Staubli VAL3: Bewegungsattribute.pjx

--- Bewegungsattribute.pjx ---
Parameters version=s7.5.3 stackSize=5000 millimeterUnit=true
Program file=MoveJoint.pgx
Program file=MoveLine.pgx
Program file=start.pgx
Program file=stop.pgx
Program file=main.pgx
Data file=Bewegungsattribute.dtx

--- Bewegungsattribute.dtx ---
frame StaubliTX240Base = {x=0.000, y=0.000, z=0.000, rx=-0.000, ry=0.000, rz=-0.000, fatherId=world[0]}
tool tCurrentTool = {x=0.000, y=0.000, z=0.000, rx=-0.000, ry=0.000, rz=-0.000, fatherId=flange[0]}
mdesc mCurrentSpeed
pointRx pPointRx1 = {}
pointRx pPointRx2 = {}

--- main.pgx ---
program main()
begin
    pPointRx1.config.shoulder = lefty
    pPointRx1.config.elbow = epositive
    pPointRx1.config.wrist = wpositive
    pPointRx2.config.shoulder = lefty
    pPointRx2.config.elbow = epositive
    pPointRx2.config.wrist = wpositive
    mCurrentSpeed.tvel = 100.00
    mCurrentSpeed.blend = joint
    mCurrentSpeed.reach = 0.010
    mCurrentSpeed.leave = 0.010
    		// Program Bewegungsattribute start
		// Program generated by RoboDK v5.2.1 for Staubli TX2-40 on 26/04/2021 13:26:34
		mCurrentSpeed.accel = 30.000
		mCurrentSpeed.decel = 30.000
		mCurrentSpeed.vel = 30.000
		mCurrentSpeed.tvel = 30.000
		mCurrentSpeed.rvel = 30.000
		link(pPointRx1,StaubliTX240Base)
		link(pPointRx2,StaubliTX240Base)
		call MoveJoint(0.00000,0.00000,90.00000,0.00000,0.00000,-0.00000)
		call MoveJoint(0.75339,44.25550,52.41940,0.00000,83.32510,0.75339)
		call MoveJoint(-10.97790,47.35230,41.99440,0.00000,90.65320,-10.97790)
		call MoveJoint(-1.36528,60.04990,34.36770,0.00000,85.58250,-1.36528)
		call MoveJoint(0.00000,0.00000,90.00000,0.00000,0.00000,-0.00000)
		mCurrentSpeed.rvel = 1000.000
		call MoveJoint(0.75339,44.25550,52.41940,0.00000,83.32510,0.75339)
		call MoveJoint(-10.97790,47.35230,41.99440,0.00000,90.65320,-10.97790)
		call MoveJoint(-1.36528,60.04990,34.36770,0.00000,85.58250,-1.36528)
		call MoveJoint(0.00000,0.00000,90.00000,0.00000,0.00000,-0.00000)
		mCurrentSpeed.tvel = 1000.000
		call MoveJoint(0.75339,44.25550,52.41940,0.00000,83.32510,0.75339)
		call MoveJoint(-10.97790,47.35230,41.99440,0.00000,90.65320,-10.97790)
		call MoveJoint(-1.36528,60.04990,34.36770,0.00000,85.58250,-1.36528)
		call MoveJoint(0.00000,0.00000,90.00000,0.00000,0.00000,-0.00000)
		mCurrentSpeed.vel = 100.000
		call MoveJoint(0.75339,44.25550,52.41940,0.00000,83.32510,0.75339)
		call MoveJoint(-10.97790,47.35230,41.99440,0.00000,90.65320,-10.97790)
		call MoveJoint(-1.36528,60.04990,34.36770,0.00000,85.58250,-1.36528)
		call MoveJoint(0.00000,0.00000,90.00000,0.00000,0.00000,-0.00000)
		mCurrentSpeed.accel = 100.000
		call MoveJoint(0.75339,44.25550,52.41940,0.00000,83.32510,0.75339)
		call MoveJoint(-10.97790,47.35230,41.99440,0.00000,90.65320,-10.97790)
		call MoveJoint(-1.36528,60.04990,34.36770,0.00000,85.58250,-1.36528)
		call MoveJoint(0.00000,0.00000,90.00000,0.00000,0.00000,-0.00000)
		mCurrentSpeed.decel = 100.000
		call MoveJoint(0.75339,44.25550,52.41940,0.00000,83.32510,0.75339)
		call MoveJoint(-10.97790,47.35230,41.99440,0.00000,90.65320,-10.97790)
		call MoveJoint(-1.36528,60.04990,34.36770,0.00000,85.58250,-1.36528)
		call MoveJoint(0.00000,0.00000,90.00000,0.00000,0.00000,-0.00000)

		waitEndMove()
		// Program Bewegungsattribute end

end

--- start.pgx ---
program start()
begin
  call main()
end

--- MoveJoint.pgx ---
program MoveJoint(num x_nJ1, num x_nJ2, num x_nJ3, num x_nJ4, num x_nJ5, num x_nJ6)
  local joint l_jJoint
begin
  l_jJoint.j1 = x_nJ1
  l_jJoint.j2 = x_nJ2
  l_jJoint.j3 = x_nJ3
  l_jJoint.j4 = x_nJ4
  l_jJoint.j5 = x_nJ5
  l_jJoint.j6 = x_nJ6
  movej(l_jJoint,tCurrentTool ,mCurrentSpeed)
end
